FUNCTION f_MessageSet : BOOL
VAR_INPUT
  stMessage     : ST_Message;
END_VAR
VAR
  _uiIndex      : UINT;
  _MainDevice   : e_Device;
  _nModRes      : UDINT;     // residual after modulo
END_VAR

stMessage.tTime                     := GVL_MSG.sLocalTime;

// why here? so all calls to this function may stay the same
_nModRes                            := stMessage.eDevice MOD e_Device.General;
_MainDevice                         := stMessage.eDevice - _nModRes;

CASE _MainDevice
OF
  e_device.DataProduct:
    // this is your data, if you choose to use this message system
    FOR _uiIndex := 1 TO GVL_MSG.MAX_MESSAGE
    DO
      IF (GVL_MSG.ProductMessages[_uiIndex].eType = e_MessageType.eMessageEmpty)
      THEN
        GVL_MSG.ProductMessages[_uiIndex]      := stMessage;
        GVL_MSG.MessageProductIndex            := _uiIndex;
        EXIT;
      END_IF
    END_FOR
  
    IF (stMessage.eType = E_MessageType.eMessageError)
    THEN
      // in case of error: increment counter
      GVL_MSG.MessageProductError     := GVL_MSG.MessageProductError + 1;
    END_IF


  e_Device.Process,
  e_Device.Application:
    FOR _uiIndex := 1 TO GVL_MSG.MAX_MESSAGE
    DO
      IF (GVL_MSG.ApplicationMessages[_uiIndex].eType = e_MessageType.eMessageEmpty)
      THEN
        GVL_MSG.ApplicationMessages[_uiIndex]  := stMessage;    // yes, we grab global values directly, only here
        GVL_MSG.MessageApplicationIndex        := _uiIndex;
        EXIT;
      END_IF
    END_FOR
    IF (stMessage.eType = E_MessageType.eMessageError)
    THEN
      // in case of error: increment counter
      GVL_MSG.MessageApplicationError := GVL_MSG.MessageApplicationError + 1;
    END_IF

  e_Device.Metrics:
    FOR _uiIndex := 1 TO GVL_MSG.MAX_MESSAGE
    DO
      IF (GVL_MSG.MetricsMessages[_uiIndex].eType = e_MessageType.eMessageEmpty)
      THEN
        GVL_MSG.MetricsMessages[_uiIndex]  := stMessage;    // yes, we grab global values directly, only here
        GVL_MSG.MessageMetricsIndex        := _uiIndex;
        EXIT;
      END_IF
    END_FOR
    IF (stMessage.eType = E_MessageType.eMessageError)
    THEN
      // in case of error: increment counter
      GVL_MSG.MessageMetricsError := GVL_MSG.MessageMetricsError + 1;
    END_IF

ELSE
  FOR _uiIndex := 1 TO GVL_MSG.MAX_MESSAGE
  DO
    IF (GVL_MSG.TransportMessages[_uiIndex].eType = e_MessageType.eMessageEmpty)
    THEN
      GVL_MSG.TransportMessages[_uiIndex]      := stMessage;
      GVL_MSG.MessageTransportIndex            := _uiIndex;
      EXIT;
    END_IF
  END_FOR

  IF (stMessage.eType = E_MessageType.eMessageError)
  THEN
    // in case of error: increment counter
    GVL_MSG.MessageTransportError := GVL_MSG.MessageTransportError + 1;
  END_IF
END_CASE

END_FUNCTION

(* stored: Version 1.1.0.1, ProductVersion 3.1.4026.13
   POU f_MessageSet: Id {7dd9a0ea-132a-4368-8b98-e527af9ed450}, SpecialFunc None *)
